// TwinCAT 3 PLC project PLC
// ProgramVersion: 3.1.4026.19
// CompilerDefines: VISU_USEPROPERTYINFO
// libraries:
//   SPT Base Types, * (Beckhoff Automation LLC)
//   SPT Components, * (Beckhoff Automation LLC)
//   SPT Diagnostic, * (Beckhoff Automation LLC)
//   SPT EtherCat, * (Beckhoff Automation LLC)
//   SPT Event Logger, * (Beckhoff Automation LLC)
//   SPT Motion Control, * (Beckhoff Automation LLC)
//   SPT Utilities, * (Beckhoff Automation LLC)
//   Tc2_Standard, * (Beckhoff Automation GmbH)
//   Tc2_System, * (Beckhoff Automation GmbH)
//   Tc3_EventLogger, * (Beckhoff Automation GmbH)
//   Tc3_PackML_V3, * (Beckhoff Automation GmbH)
// project tree:
//   Components/ Component.TcPOU
//   / GlobalTextList.TcGTLO, PlcTask.TcTTO, Visualization Manager.TcVMO (not stored)
//   Modules/00 Machine/ Machine.TcPOU
//   Modules/01 Infeed/ Infeed.TcPOU
//   POUs/ MAIN.TcPOU
//   VISUs/ Visualization.TcVIS
// real-time tasks:
//   TASK PlcTask: cycle T#10ms, priority 20, ADS port 350

CONFIGURATION PLC
    RESOURCE PLC ON TwinCAT3
        TASK PlcTask(INTERVAL := T#10ms, PRIORITY := 20);
        PROGRAM MAIN WITH PlcTask : MAIN;
    END_RESOURCE
END_CONFIGURATION

// ---- POUs/MAIN.TcPOU
PROGRAM MAIN
VAR
	Machine : Machine := (Name := 'Machine');
END_VAR

// All sample code provided by Beckhoff Automation LLC are for illustrative purposes only and are provided “as is” and without any warranties, express or implied. Actual implementations in applications will vary significantly. Beckhoff Automation LLC shall have no liability for, and does not waive any rights in relation to, any code samples that it provides or the use of such code samples for any purpose.

//
Machine.CyclicLogic();

(*
	This sample demonstrates the reactions of the state machine based on the _ParentFaultResponseDefinitions.
	
The _ParentFaultResponseDefinitions exists for all inherited classes of FB_PackML_BaseModule and FB_ComponentBase.
This allows for the class that raises the Error to dictate the response of the upper-level code (EM or MM) that is monitoring it.
                
When an event happens, it will be logged in the Error List of the IDE under Errors, Warnings, or Messages.
The _ParentFaultResponseDefinitions for each specific TcEventSeverity will determine how the upper-level Parent Module will respond.
                
The default response for TcEventSeverity.Error and TcEventSeverity.Critical is E_AlarmResponse.Abort_ImmediateError.
This will cause the Parent Module to command itself into the Aborting state and also raise an error that will set its own _CurrentAlarmSeverity to Error.
This in turn will result in its Parent Module repeating the process of logging an error, issuing itself an Abort command and setting its own _CurrentAlarmSeverity to Error.


If a Component set its _ParentFaultResponseDefinitions[TcEventSeverity.Error] to E_AlarmResponse.Abort_Immediate then its Parent Module will not log an error, 
but instead log a warning, set its _CurrentAlarmSeverity to Warning and issue itself an Abort command.

Because the default response to a Warning is NoResponse the Machine Module will not respond to the parent module of the faulted component having a _CurrentAlarmSeverity of Warning.
	
	
If you want the MM to Abort along with the EM when a Component raises an Error you must control the value of _CurrentAlarmSeverity. 

	In the CyclicLogic method of the MM the _CurrentAlarmSeverity is updated by the following:
		1.	Super^.CyclicLogic resets the _CurrentAlarmSeverity to Verbose
		2.	_CurrentAlarmSeverity is updated based on the Alarms of the EM
	
	Code can be added to update the _CurrentAlarmSeverity of the EM based on the _CurrentAlarmSeverity of its Components
	Set _ParentFaultResponseDefinitions[TcEventSeverity.Error] := E_AlarmResponse.Abort_Immediate; for the EM and the Components 
	Then add the code to the CyclicLogic to read the _CurrentAlarmSeverity of the Components of the EM, this will give an Error message only for the Component that raises an Error, but still cause the EM and MM to go into Abort.
	See the Infeed.CyclicLogic() method for an example.


Using the Visu to test reactions:
	
The Warning and Error definitions are set to their defaults on startup, for the MM, EM, and Component

_ParentFaultResponseDefinitions[TcEventSeverity.Warning] := E_AlarmResponse.NoResponse;
_ParentFaultResponseDefinitions[TcEventSeverity.Error] := E_AlarmResponse.Abort_ImmediateError;

The Visualization provides buttons to toggle an Error. When the error is raised the state machine of the EM and MM will respond according to the selected _ParentFaultResponseDefinitions.

Default Configuration:
The default response is for the Component log its error and set its CurrentSeverity to Error. 
The EM is monitoring the Component and will respond to the CurrentSeverity of Error by changing its State Command to Abort.
The EM will log the error and set its CurrentSeverity to Error.
The MM is monitoring the EM and will respond to the CurrentSeverity of Error by changing its State Command to Abort.
The MM will log the error and set its CurrentSeverity to Error.

This causes a single error in a component to generate 3 messages in the Error List.

Muting Component Errors:
If the _ParentFaultResponseDefinitions[TcEventSeverity.Error] for the Component is changed from E_AlarmResponse.Abort_ImmediateError to E_AlarmResponse.Abort_Immediate
then the EM that is monitoring the Component will set its Current Severity to Warning and only the Component will log an error.
The EM will abort becuase its Component has an Error, but the MM will not abort because its EM's Current Severity is Warning.

If the 	_ParentFaultResponseDefinitions[TcEventSeverity.Error] for the Component is set to E_AlarmResponse.NoResponse
then the Component will log its error and set its Current Severity to Error. But the EM will not respond, change its state or its CurrentSeverity.

If the	_ParentFaultResponseDefinitions[TcEventSeverity.Error] for the Component is left at E_AlarmResponse.Abort_ImmediateError
and the _ParentFaultResponseDefinitions[TcEventSeverity.Error] for the EM is set to E_AlarmResponse.Abort_Immediate
then the Component and EM will both write to the log, and both 'Parents' (EM and MM) will Abort.
	


*)

END_PROGRAM

// ---- Modules/00 Machine/Machine.TcPOU
FUNCTION_BLOCK Machine EXTENDS FB_PackML_BaseModule
VAR
	Infeed			 : Infeed := (Name := 'Infeed');
	_ErrorSeverity	 : INT	  := 2;
	_WarningSeverity : INT;
END_VAR

METHOD ChangeAlarmSeverity
CASE _WarningSeverity OF
	0:
		_ParentFaultResponseDefinitions[TcEventSeverity.Warning] := E_AlarmResponse.NoResponse;

	1:
		_ParentFaultResponseDefinitions[TcEventSeverity.Warning] := E_AlarmResponse.Abort_Immediate;

	2:
		_ParentFaultResponseDefinitions[TcEventSeverity.Warning] := E_AlarmResponse.Abort_ImmediateError;
END_CASE

CASE _ErrorSeverity OF
	0:
		_ParentFaultResponseDefinitions[TcEventSeverity.Error] := E_AlarmResponse.NoResponse;

	1:
		_ParentFaultResponseDefinitions[TcEventSeverity.Error] := E_AlarmResponse.Abort_Immediate;

	2:
		_ParentFaultResponseDefinitions[TcEventSeverity.Error] := E_AlarmResponse.Abort_ImmediateError;
END_CASE
END_METHOD

METHOD CyclicLogic
IF NOT _InitComplete THEN
	_InitComplete := Initialize();
	RETURN;
END_IF

//
ChangeAlarmSeverity();
SUPER^.CyclicLogic();
END_METHOD

(* Automatically enables and disables HMI control based on the PackML mode*)
METHOD PROTECTED HMIPermissions
AllowHMIControl(TRUE);
END_METHOD

(* Basic module initialization logic*)
METHOD PROTECTED Initialize : BOOL
Initialize := FALSE;
CASE DescendantSequenceState OF
	0:
		LogModeChanges	:= FALSE;
		LogStateChanges := FALSE;

		//
		RegisterSubmodule(SubModule := Infeed);
		DescendantSequenceState := DescendantSequenceState + 10;

	10:
		_ParentFaultResponseDefinitions[TcEventSeverity.Error] := E_AlarmResponse.Abort_ImmediateError;
		DescendantSequenceState								   := DescendantSequenceState + 10;

	20:
		IF SUPER^.Initialize() THEN
			DescendantSequenceState := DescendantSequenceState + 10;
		END_IF

	30:
		Initialize := TRUE;
END_CASE
END_METHOD

END_FUNCTION_BLOCK

// ---- Modules/01 Infeed/Infeed.TcPOU
FUNCTION_BLOCK Infeed EXTENDS FB_PackML_BaseModule
VAR
	Component		 : Component := (Name := 'Component');
	InfeedAlarms	 : ARRAY[1..INFEED_ALARM_COUNT] OF FB_TcAlarm;
	testError		 : BOOL;
	_ErrorSeverity	 : INT := 2;
	_WarningSeverity : INT;
	Axis			 : FB_Component_BasicAxis;
END_VAR

VAR CONSTANT
	INFEED_ALARM_COUNT : UDINT := 6; //First is InitReferenceEvent
END_VAR

METHOD ChangeAlarmSeverity
CASE _WarningSeverity OF
	0:
		_ParentFaultResponseDefinitions[TcEventSeverity.Warning] := E_AlarmResponse.NoResponse;

	1:
		_ParentFaultResponseDefinitions[TcEventSeverity.Warning] := E_AlarmResponse.Abort_Immediate;

	2:
		_ParentFaultResponseDefinitions[TcEventSeverity.Warning] := E_AlarmResponse.Abort_ImmediateError;
END_CASE

CASE _ErrorSeverity OF
	0:
		_ParentFaultResponseDefinitions[TcEventSeverity.Error] := E_AlarmResponse.NoResponse;

	1:
		_ParentFaultResponseDefinitions[TcEventSeverity.Error] := E_AlarmResponse.Abort_Immediate;

	2:
		_ParentFaultResponseDefinitions[TcEventSeverity.Error] := E_AlarmResponse.Abort_ImmediateError;
END_CASE
END_METHOD

METHOD PROTECTED Clearing
F_ClearAllEventsInClass(Alarms := InfeedAlarms);
SUPER^.Clearing();
END_METHOD

(* Initializes event function blocks using this module's name*)
METHOD PROTECTED CreateEvents
F_CreateAllEventsInClass(Alarms		:= InfeedAlarms,
						 ClassSize	:= SIZEOF(TC_Events.Events_Infeed),
						 pInitEvent := ADR(TC_EVENTS.Events_Infeed.InitReferenceEvent),
						 Prefix		:= Name);

SUPER^.CreateEvents();
END_METHOD

METHOD CyclicLogic
VAR
	i : UDINT;
END_VAR
IF NOT _InitComplete THEN
	_InitComplete := Initialize();
	RETURN;
END_IF

//
ChangeAlarmSeverity();
EventMonitor();
SUPER^.CyclicLogic();

(*
*
*		Code must be after SUPER^.CyclicLogic();
*
*)

(* Update alarm severity from this module *)
_CurrentAlarmSeverity := F_GetMaxSeverityRaised(Alarms := InfeedAlarms, CurrentSeverity := _CurrentAlarmSeverity);

// Add this code to set the _CurrentAlarmSeverity for this EM to match the highest _CurrentAlarmSeverity of its Components.

//Update alarm severity for this module to match the highest EventSeverity of all Components
FOR i := 1 TO NumberOfComponents DO
	IF ipComponents[i].CurrentAlarmSeverity >= TcEventSeverity.Error THEN
		_CurrentAlarmSeverity := TcEventSeverity.Error;
	END_IF
END_FOR

//
_Error := _CurrentAlarmSeverity >= TcEventSeverity.Error;
END_METHOD

METHOD EventMonitor
VAR_INPUT
END_VAR
IF testError AND_THEN NOT InfeedAlarms[E_Events_Infeed.Error].bRaised THEN
	RaiseAlarm2Args(InfeedAlarms[E_Events_Infeed.Error], 'Note 1', 'Note 2');
END_IF
END_METHOD

(* Basic module initialization logic*)
METHOD PROTECTED Initialize : BOOL
VAR
END_VAR
Initialize := FALSE;
CASE DescendantSequenceState OF
	0:
		LogModeChanges	:= FALSE;
		LogStateChanges := FALSE;

		//
		RegisterComponent(Component := Component);
		DescendantSequenceState := DescendantSequenceState + 10;

	10:
		_ParentFaultResponseDefinitions[TcEventSeverity.Warning] := E_AlarmResponse.NoResponse;
		_ParentFaultResponseDefinitions[TcEventSeverity.Error]	 := E_AlarmResponse.Abort_ImmediateError;
		DescendantSequenceState									 := DescendantSequenceState + 10;

	20:
		IF SUPER^.Initialize() THEN
			DescendantSequenceState := DescendantSequenceState + 10;
		END_IF

	30:
		Initialize := TRUE;
END_CASE
END_METHOD

METHOD RaiseAlarm2Args
VAR_IN_OUT
	Alarm : FB_TcAlarm; //Alarm to be raised
END_VAR

VAR_INPUT
	String_1 : STRING; //First String Parameter (The Name of this component will be applied first automatically)
	String_2 : STRING; //Second String Parameter
END_VAR
F_RaiseAlarmWithStringParameters(Alarm	  := Alarm,
								 String_1 := Name,
								 String_2 := String_1,
								 String_3 := String_2);
END_METHOD

END_FUNCTION_BLOCK

// ---- Components/Component.TcPOU
FUNCTION_BLOCK Component EXTENDS FB_ComponentBase
VAR
	ComponentAlarms	 : ARRAY[1..COMPONENT_ALARM_COUNT] OF FB_TcAlarm;
	testError		 : BOOL;
	_ErrorSeverity	 : INT := 2;
	_WarningSeverity : INT;
END_VAR

VAR CONSTANT
	COMPONENT_ALARM_COUNT : UDINT := 7; //First is InitReferenceEvent
END_VAR

METHOD ChangeAlarmSeverity
CASE _WarningSeverity OF
	0:
		_ParentFaultResponseDefinitions[TcEventSeverity.Warning] := E_AlarmResponse.NoResponse;

	1:
		_ParentFaultResponseDefinitions[TcEventSeverity.Warning] := E_AlarmResponse.Abort_Immediate;

	2:
		_ParentFaultResponseDefinitions[TcEventSeverity.Warning] := E_AlarmResponse.Abort_ImmediateError;
END_CASE

CASE _ErrorSeverity OF
	0:
		_ParentFaultResponseDefinitions[TcEventSeverity.Error] := E_AlarmResponse.NoResponse;

	1:
		_ParentFaultResponseDefinitions[TcEventSeverity.Error] := E_AlarmResponse.Abort_Immediate;

	2:
		_ParentFaultResponseDefinitions[TcEventSeverity.Error] := E_AlarmResponse.Abort_ImmediateError;
END_CASE
END_METHOD

// Initializes event function blocks using this components's name
METHOD PROTECTED CreateEvents

// This method is called by Initialize() as required
F_CreateAllEventsInClass(Alarms		:= ComponentAlarms,
						 ClassSize	:= SIZEOF(TC_Events.Events_Component),
						 pInitEvent := ADR(TC_EVENTS.Events_Component.InitReferenceEvent),
						 Prefix		:= Name);

SUPER^.CreateEvents();
END_METHOD

// This method serves as the entry point for all underlying FB logic
METHOD PUBLIC CyclicLogic

// This method should be called cyclically by descendant function blocks by invoking SUPER^.CyclicLogic().  Alternatively, the contents of this method could be reimplemented entirely in which case a call to this method would not be necessary.
IF NOT _InitComplete THEN
	_InitComplete := Initialize();
	RETURN;
END_IF

//
ChangeAlarmSeverity();
SUPER^.CyclicLogic();

(*
*
*		Code must be after SUPER^.CyclicLogic();
*
*)

// Update alarm severity for this component
_CurrentAlarmSeverity := F_GetMaxSeverityRaised(Alarms := ComponentAlarms, CurrentSeverity := _CurrentAlarmSeverity);
_Error				  := _CurrentAlarmSeverity >= TcEventSeverity.Error;
END_METHOD

// Provides basic error detection and event handling for this component
METHOD PROTECTED Monitoring

//This method is called cyclically by CyclicLogic()
_Busy := FALSE;

//AlarmMonitoring
IF testError AND NOT ComponentAlarms[E_Events_Component.Error].bRaised THEN
	RaiseAlarm2Args(ComponentAlarms[E_Events_Component.Error], 'Note 1', 'Note 2');
END_IF

SUPER^.Monitoring();
END_METHOD

METHOD RaiseAlarm2Args
VAR_IN_OUT
	Alarm : FB_TcAlarm; //Alarm to be raised
END_VAR

VAR_INPUT
	String_1 : STRING; //First String Parameter (The Name of this component will be applied first automatically)
	String_2 : STRING; //Second String Parameter
END_VAR
F_RaiseAlarmWithStringParameters(Alarm	  := Alarm,
								 String_1 := Name,
								 String_2 := String_1,
								 String_3 := String_2);
END_METHOD

// Clears error flags and error IDs for this component
METHOD PUBLIC Reset : BOOL

//Typically called by the EMs SUPER^.Clearing Method
F_ClearAllEventsInClass(Alarms := ComponentAlarms);
IF SUPER^.Reset() THEN
	_Error	 := FALSE;
	_ErrorID := 0;
	Reset	 := TRUE;
END_IF
END_METHOD

END_FUNCTION_BLOCK

// ---- GlobalTextList.TcGTLO
TEXTLIST GlobalTextList
  698 = '%s'
  703 = 'Abort Immediate'
  325 = 'Abort Immediate Error'
  112 = 'Alarm Severity: Error'
  69 = 'Alarm Severity: Warning'
  265 = 'Component'
  385 = 'Component Alarm'
  886 = 'Component Error'
  561 = 'Current Severity'
  793 = 'Infeed'
  952 = 'Infeed Alarm'
  47 = 'Infeed Error'
  725 = 'Machine'
  313 = 'Warning'
END_TEXTLIST

// ---- VISUs/Visualization.TcVIS
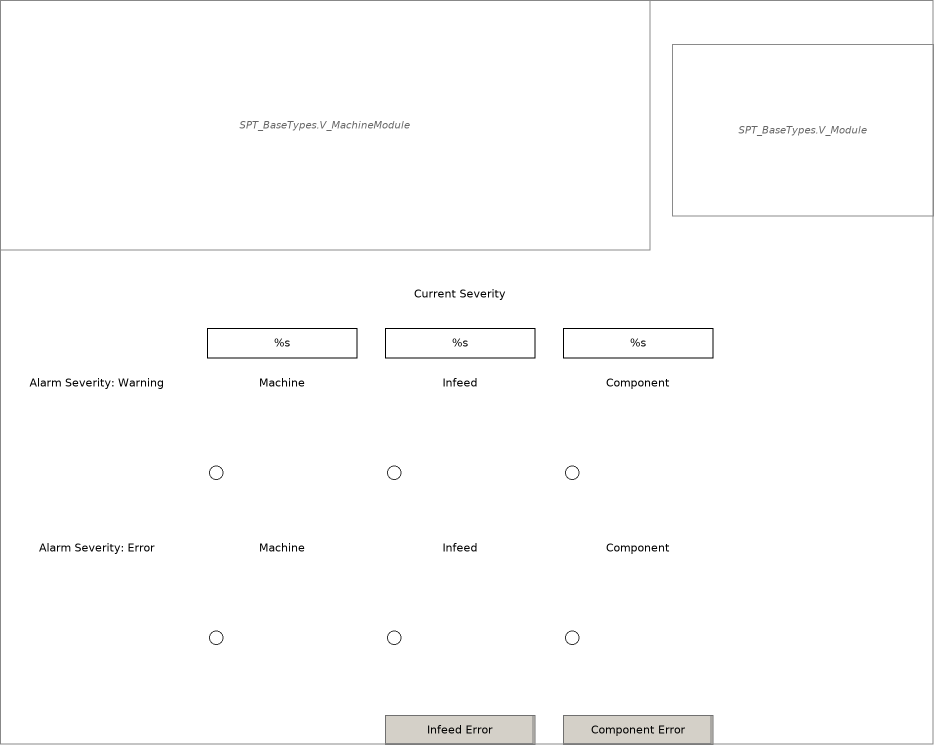
VISUALIZATION Visualization  // 934x745
    Frame (0,0 650x250)
        shows SPT_BaseTypes.V_MachineModule(HMI := MAIN.Machine.PackMLBaseModule_HMI)
    Label (207,533 150x30), "Machine"
    Label (385,533 150x30), "Infeed"
    Label (563,533 150x30), "Component"
    Label (22,533 150x30), "Alarm Severity: Error"
    RadioButton (207,584 168x107), variable: MAIN.Machine._ErrorSeverity
        Areas[0]: Text=Warning
        Areas[1]: Text=Abort Immediate
        Areas[2]: Text=Abort Immediate Error
    RadioButton (385,584 168x107), variable: MAIN.Machine.Infeed._ErrorSeverity
        Areas[0]: Text=Warning
        Areas[1]: Text=Abort Immediate
        Areas[2]: Text=Abort Immediate Error
    RadioButton (563,584 168x107), variable: MAIN.Machine.Infeed.Component._ErrorSeverity
        Areas[0]: Text=Warning
        Areas[1]: Text=Abort Immediate
        Areas[2]: Text=Abort Immediate Error
    Button (563,715 150x30), "Component Error"
        toggle MAIN.Machine.Infeed.Component.testError
    Frame (672,44 262x172)
        shows SPT_BaseTypes.V_Module(HMI := MAIN.Machine.Infeed.PackMLBaseModule_HMI)
    Button (385,715 150x30), "Infeed Error"
        toggle MAIN.Machine.Infeed.testError
    Label (207,368 150x30), "Machine"
    Label (385,368 150x30), "Infeed"
    Label (563,368 150x30), "Component"
    Label (22,368 150x30), "Alarm Severity: Warning"
    RadioButton (207,419 168x107), variable: MAIN.Machine._WarningSeverity
        Areas[0]: Text=Warning
        Areas[1]: Text=Abort Immediate
        Areas[2]: Text=Abort Immediate Error
    RadioButton (385,419 168x107), variable: MAIN.Machine.Infeed._WarningSeverity
        Areas[0]: Text=Warning
        Areas[1]: Text=Abort Immediate
        Areas[2]: Text=Abort Immediate Error
    RadioButton (563,419 168x107), variable: MAIN.Machine.Infeed.Component._WarningSeverity
        Areas[0]: Text=Warning
        Areas[1]: Text=Abort Immediate
        Areas[2]: Text=Abort Immediate Error
    Rectangle (207,328 150x30), "%s", text variable: MAIN.Machine._CurrentAlarmSeverity
    Rectangle (385,328 150x30), "%s", text variable: MAIN.Machine.Infeed._CurrentAlarmSeverity
    Rectangle (563,328 150x30), "%s", text variable: MAIN.Machine.Infeed.Component._CurrentAlarmSeverity
    Label (385,279 150x30), "Current Severity"
END_VISUALIZATION
